FUNCTION_BLOCK Trigger
VAR_INPUT
	iTRIG:	BOOL;
END_VAR
VAR_OUTPUT
	Q:	BOOL;
END_VAR
VAR
	R_TRIG_Ein:	R_TRIG;
	R_TRIG_Quit:	R_TRIG;
	F_TRIG_Ein:	F_TRIG;


	F_TRIG_Quit: F_TRIG;
END_VAR

(* Abfrage des Ereignisses auf Flanke und Quittung zur Wiederholung der Meldung *)

R_TRIG_Ein	(CLK := (iTRIG));
F_TRIG_Ein	(CLK := (iTRIG));
//R_TRIG_Quit	(CLK := LS_RW.OBJ65101.Quit_1s);
F_TRIG_Quit	(CLK := stPecomRW.OBJ_RW_65101.Quit_1s  AND iTRIG );

Q := R_TRIG_EIN.Q OR F_TRIG_EIN.Q OR R_TRIG_Quit.Q OR F_TRIG_Quit.Q;

END_FUNCTION_BLOCK

(* stored: Version 1.1.0.1, ProductVersion 3.1.4024.12
   POU Trigger: Id {bdebb5ef-c840-4239-92a8-81b80e9657ae}, SpecialFunc None *)
